# B&R Automation Studio project YuMiLAB_project (part 2)

#### Main.c
```c
// ************************************************************************************************************************************ //
// Title: Data processing -> Barcode Scanner
// Autor: Roman Parak
// Date : 8.5.2020
// Email: Roman.Parak@outlook.com
// ************************************************************************************************************************************ //

// ************************************************************************************************************************************ //
// -------------------------------------------------------------  LIBRARIES ----------------------------------------------------------- //
// ************************************************************************************************************************************ //
#include <bur/plctypes.h>

#ifdef _DEFAULT_INCLUDES
	#include <AsDefault.h>
#endif

#include <astime.h>

// ************************************************************************************************************************************ //
// -------------------------------------------------------------  DECLARATIONS -------------------------------------------------------- //
// ************************************************************************************************************************************ //
// BOOL
_LOCAL BOOL enable;
// UINT
_LOCAL UINT status;
_LOCAL UINT barcode_state;
// DATE_AND_TIME
_LOCAL DATE_AND_TIME DT1;
// DTGetTime_typ
_LOCAL DTGetTime_typ DTGetTime_1;
// INT
_LOCAL INT scan_counter;

// Declaration functions
void reset_data_mv();
void reset_data_init();

// ************************************************************************************************************************************ //
// -----------------------------------------------------------  INITIALIZATION -------------------------------------------------------- //
// ************************************************************************************************************************************ //
void _INIT ProgramInit(void)
{
	// Read/Write Data from Rpi
	(UDINT)strcpy(g_YuMiLab.scanner_m.rw_data_barcode.barcode_id, "");
	(UDINT)strcpy(g_YuMiLab.scanner_m.rw_data_barcode.tray_id, "");

	// Barcode parameters
	g_YuMiLab.scanner_m.rw_data_barcode.command    = 0;
	g_YuMiLab.scanner_m.rw_data_barcode.error_code = 0;
	g_YuMiLab.scanner_m.rw_data_barcode.barcode_scanner_module_ok = 0;
	g_YuMiLab.scanner_m.rw_data_barcode.tray_position_column = 3;
	g_YuMiLab.scanner_m.rw_data_barcode.tray_position_row    = 4;

	// Actual Data
	(UDINT)strcpy(g_YuMiLab.scanner_m.actual_barcode_id, "");
	(UDINT)strcpy(g_YuMiLab.scanner_m.actual_tray_id, "");

	// Data MappView {history} -> Initialization
	reset_data_mv();

	// FeID set/reset
	g_YuMiLab.scanner_m.feid_cmd_str.set = 0;
	g_YuMiLab.scanner_m.feid_cmd_str.reset = 0;
	g_YuMiLab.scanner_m.feid_cmd_str.enable_mv = 1;

	// Feid command
	(UDINT)strcpy(g_YuMiLab.scanner_m.feid_cmd_str.tray_id,"");

	// Main State
	barcode_state = 0;

	// Scan counter
	scan_counter = 0;
}

// ************************************************************************************************************************************ //
// -----------------------------------------------------------  MAIN (Cyclic) --------------------------------------------------------- //
// ************************************************************************************************************************************ //
void _CYCLIC ProgramCyclic(void)
{

	switch(barcode_state){
		case 0:
			{
				/*************************************** INITIALIZATION STATE ******************************************/

				// err-states:
				/*
				ok = 0
				eID_not_in_database = 1
				tray_warning_FeID_used = 2  # no new DB entry added for sample_tray, using existing
				tray_not_created = 3  # cannot add new sample_tray
				tray_position_not_assigned = 4
				service_connection_lost = 5  # cannot access DB
				*/
				// cmd {0} -> nothing ok, cmd {1} - write FeID , cmd {2} -> scan, cmd {3} ->  write row, column

				//(UDINT)strcpy(g_YuMiLab.scanner_m.rw_data_barcode.barcode_id, "");

				// reset scan err.
				g_YuMiLab.scanner_m.scan_err = 0;

				// Copy
				g_YuMiLab.scanner_m.cmd.write_FeID = g_YuMiLab.scanner_m.feid_cmd_str.set;

				// Condition -> Scanner module is ok!
				if(g_YuMiLab.scanner_m.rw_data_barcode.barcode_scanner_module_ok == 1){
					// reset error code
					g_YuMiLab.scanner_m.rw_data_barcode.error_code = 0;

					if(g_YuMiLab.scanner_m.cmd.write_FeID == 1){
						//cmd {1} - write FeID
						barcode_state = 1;
					}else if(g_YuMiLab.scanner_m.cmd.scan == 1){
						//cmd {2} -> scan
						(UDINT)strcpy(g_YuMiLab.scanner_m.rw_data_barcode.barcode_id, "None");
						// change state
						barcode_state = 3;
					}
				}
			}
			break;

		case 1:
			{
				/*************************************** WRITE FEID (1) STATE ******************************************/
				// reset write (Feid) command
				g_YuMiLab.scanner_m.cmd.write_FeID = 0;

				// mappview -> enable
				g_YuMiLab.scanner_m.feid_cmd_str.enable_mv = 0;

				// copy string
				(UDINT)strcpy(g_YuMiLab.scanner_m.actual_tray_id ,g_YuMiLab.scanner_m.feid_cmd_str.tray_id);
				(UDINT)strcpy(g_YuMiLab.scanner_m.rw_data_barcode.tray_id,g_YuMiLab.scanner_m.feid_cmd_str.tray_id);

				// command set -> 1
				g_YuMiLab.scanner_m.rw_data_barcode.command = 1;

				// change state -> check result
				barcode_state = 2;

			}
			break;
		case 2:
			{
				/*************************************** WRITE FEID (1a) STATE ******************************************/
				// Err. Condition -> module, err. code -> see bellow (info)
				if(g_YuMiLab.scanner_m.rw_data_barcode.barcode_scanner_module_ok == 0 || g_YuMiLab.scanner_m.rw_data_barcode.error_code > 0){
					// err. state var.
					err_state_barcode = 1;
					// command -> null
					g_YuMiLab.scanner_m.rw_data_barcode.command = 0;
					// change state -> initialization
					barcode_state = 0;
				}

				// Condition -> cmd null
				if(g_YuMiLab.scanner_m.rw_data_barcode.command == 0){
					// change state -> initialization
					barcode_state = 0;
				}
			}
			break;
		case 3:
			{
				/*************************************** START SCAN (1) STATE ******************************************/

				// scan var. -> null
				g_YuMiLab.scanner_m.cmd.scan = 0;

				// command -> 2
				g_YuMiLab.scanner_m.rw_data_barcode.command = 2;

				// changa state
				barcode_state = 4;

				// Err. Condition -> module
				if(g_YuMiLab.scanner_m.rw_data_barcode.barcode_scanner_module_ok == 0){
					// err. state var.
					err_state_barcode = 1;
					// command -> null
					g_YuMiLab.scanner_m.rw_data_barcode.command = 0;
					// change state -> initialization
					barcode_state = 0;
				}
			}
			break;

		case 4:
			{
				/*************************************** START SCAN (1a) STATE ******************************************/

				if(g_YuMiLab.scanner_m.rw_data_barcode.command == 0){
					//cmd {3} -> write row, column
					barcode_state = 5;
				}else if(g_YuMiLab.scanner_m.rw_data_barcode.error_code > 0 || (barcode_scan_state_next == 1 && g_YuMiLab.scanner_m.rw_data_barcode.command > 0)){
					// Err. Condition -> module, err. code -> see bellow (info)
					// err. state var.
					err_state_barcode = 1;
					// command -> null
					g_YuMiLab.scanner_m.rw_data_barcode.command = 0;

					// continue
					barcode_state = 5;
				}
			}
			break;
		case 5:
			{
				/*************************************** START SCAN (2) STATE ******************************************/

				// read barcode id
				(UDINT)strcpy(g_YuMiLab.scanner_m.actual_barcode_id , g_YuMiLab.scanner_m.rw_data_barcode.barcode_id);
				// write to table
				(UDINT)strcpy(g_YuMiLab.scanner_m.data_mv.barcode_id[scan_counter],g_YuMiLab.scanner_m.rw_data_barcode.barcode_id);
				// write column, row -> index of the current barcode ID
				g_YuMiLab.scanner_m.rw_data_barcode.tray_position_column = g_YuMiLab.scanner_m.data_mv.index_column[scan_counter];
				g_YuMiLab.scanner_m.rw_data_barcode.tray_position_row    = g_YuMiLab.scanner_m.data_mv.index_row[scan_counter];

				// Get actual time
				DTGetTime_1.enable = 1;
				// Call function
				DTGetTime(&DTGetTime_1);
				// Write time to the table
				ascDT(DTGetTime_1.DT1,(UDINT)&g_YuMiLab.scanner_m.data_mv.time[scan_counter], 128);

				// turn off function block
				DTGetTime_1.enable = 0;

				// Err. Condition -> err. code
				if(g_YuMiLab.scanner_m.rw_data_barcode.error_code > 0){
					// err. state var.
					err_state_barcode = 1;
					// error info -> with current index
					g_YuMiLab.scanner_m.data_mv.err_info[scan_counter] = 1;
				}

				// command -> 3
				g_YuMiLab.scanner_m.rw_data_barcode.command = 3;

				// change state
				barcode_state = 6;

			}
			break;

		case 6:
			{
				/*************************************** START SCAN (3) STATE ******************************************/

				// Err. Condition -> module, err. code -> see bellow (info)
				if(g_YuMiLab.scanner_m.rw_data_barcode.barcode_scanner_module_ok == 0 || g_YuMiLab.scanner_m.rw_data_barcode.error_code > 0){
					// err. state var.
					err_state_barcode = 1;

					// check counter max var.
					if(scan_counter < 11){
						// increase var. + 1
						scan_counter = scan_counter + 1;
					}else {
						// reset counter
						scan_counter = 0;
					}

					// command -> null
					g_YuMiLab.scanner_m.rw_data_barcode.command = 0;

					// change state -> initialization
					barcode_state = 0;
				}else{

					// Condition -> Command null (info from barcode app.)?
					if(g_YuMiLab.scanner_m.rw_data_barcode.command == 0){
						// check counter max var.
						if(scan_counter < 11){
							// increase var. + 1
							scan_counter = scan_counter + 1;
						}else {
							// reset counter
							scan_counter = 0;
						}

						// change state -> initialization
						barcode_state = 0;
					}else if(barcode_scan_state_next == 1 && g_YuMiLab.scanner_m.rw_data_barcode.command > 0){
						// Condition -> Command > 0 (no information from barcode app.) and aux. var from another task (Robot_m.c)
						// err. state var.
						err_state_barcode = 1;
						// command -> null
						g_YuMiLab.scanner_m.rw_data_barcode.command = 0;

						// check counter max var.
						if(scan_counter < 11){
							// increase var. + 1
							scan_counter = scan_counter + 1;
						}else {
							// reset counter
							scan_counter = 0;
						}

						// change state -> initialization
						barcode_state = 0;
					}
				}

				// Copy counter: Local var. -> Global var.
				g_YuMiLab.robot_m.counter = scan_counter;
			}
			break;
	}

	// function for reset current Feid
	if(g_YuMiLab.scanner_m.feid_cmd_str.reset == 1){
		// Feid -> null
		(UDINT)strcpy(g_YuMiLab.scanner_m.feid_cmd_str.tray_id,"");
		// enable textbox
		g_YuMiLab.scanner_m.feid_cmd_str.enable_mv = 1;
	}

	// reset mappview data
	if(g_YuMiLab.scanner_m.reset_data_mv == 1){
		// call function
		reset_data_init();
	}
}

// ************************************************************************************************************************************ //
// ------------------------------------------------------------  FUNCTIONS ------------------------------------------------------------ //
// ************************************************************************************************************************************ //

// **************** RESET DATA MAPPVIEW ********************** //
void reset_data_mv(){
	(UDINT)strcpy(g_YuMiLab.scanner_m.data_mv.barcode_id[0], "");
	(UDINT)strcpy(g_YuMiLab.scanner_m.data_mv.barcode_id[1], "");
	(UDINT)strcpy(g_YuMiLab.scanner_m.data_mv.barcode_id[2], "");
	(UDINT)strcpy(g_YuMiLab.scanner_m.data_mv.barcode_id[3], "");
	(UDINT)strcpy(g_YuMiLab.scanner_m.data_mv.barcode_id[4], "");
	(UDINT)strcpy(g_YuMiLab.scanner_m.data_mv.barcode_id[5], "");
	(UDINT)strcpy(g_YuMiLab.scanner_m.data_mv.barcode_id[6], "");
	(UDINT)strcpy(g_YuMiLab.scanner_m.data_mv.barcode_id[7], "");
	(UDINT)strcpy(g_YuMiLab.scanner_m.data_mv.barcode_id[8], "");
	(UDINT)strcpy(g_YuMiLab.scanner_m.data_mv.barcode_id[9], "");
	(UDINT)strcpy(g_YuMiLab.scanner_m.data_mv.barcode_id[10], "");
	(UDINT)strcpy(g_YuMiLab.scanner_m.data_mv.barcode_id[11], "");

	(UDINT)strcpy(g_YuMiLab.scanner_m.data_mv.time[0], "");
	(UDINT)strcpy(g_YuMiLab.scanner_m.data_mv.time[1], "");
	(UDINT)strcpy(g_YuMiLab.scanner_m.data_mv.time[2], "");
	(UDINT)strcpy(g_YuMiLab.scanner_m.data_mv.time[3], "");
	(UDINT)strcpy(g_YuMiLab.scanner_m.data_mv.time[4], "");
	(UDINT)strcpy(g_YuMiLab.scanner_m.data_mv.time[5], "");
	(UDINT)strcpy(g_YuMiLab.scanner_m.data_mv.time[6], "");
	(UDINT)strcpy(g_YuMiLab.scanner_m.data_mv.time[7], "");
	(UDINT)strcpy(g_YuMiLab.scanner_m.data_mv.time[8], "");
	(UDINT)strcpy(g_YuMiLab.scanner_m.data_mv.time[9], "");
	(UDINT)strcpy(g_YuMiLab.scanner_m.data_mv.time[10], "");
	(UDINT)strcpy(g_YuMiLab.scanner_m.data_mv.time[11], "");

	g_YuMiLab.scanner_m.data_mv.err_info[0] = 0;
	g_YuMiLab.scanner_m.data_mv.err_info[1] = 0;
	g_YuMiLab.scanner_m.data_mv.err_info[2] = 0;
	g_YuMiLab.scanner_m.data_mv.err_info[3] = 0;
	g_YuMiLab.scanner_m.data_mv.err_info[4] = 0;
	g_YuMiLab.scanner_m.data_mv.err_info[5] = 0;
	g_YuMiLab.scanner_m.data_mv.err_info[6] = 0;
	g_YuMiLab.scanner_m.data_mv.err_info[7] = 0;
	g_YuMiLab.scanner_m.data_mv.err_info[8] = 0;
	g_YuMiLab.scanner_m.data_mv.err_info[9] = 0;
	g_YuMiLab.scanner_m.data_mv.err_info[10] = 0;
	g_YuMiLab.scanner_m.data_mv.err_info[11] = 0;

	g_YuMiLab.scanner_m.data_mv.index[0] = 1;
	g_YuMiLab.scanner_m.data_mv.index[1] = 2;
	g_YuMiLab.scanner_m.data_mv.index[2] = 3;
	g_YuMiLab.scanner_m.data_mv.index[3] = 4;
	g_YuMiLab.scanner_m.data_mv.index[4] = 5;
	g_YuMiLab.scanner_m.data_mv.index[5] = 6;
	g_YuMiLab.scanner_m.data_mv.index[6] = 7;
	g_YuMiLab.scanner_m.data_mv.index[7] = 8;
	g_YuMiLab.scanner_m.data_mv.index[8] = 9;
	g_YuMiLab.scanner_m.data_mv.index[9] = 10;
	g_YuMiLab.scanner_m.data_mv.index[10] = 11;
	g_YuMiLab.scanner_m.data_mv.index[11] = 12;

	g_YuMiLab.scanner_m.data_mv.index_column[0] = 1;
	g_YuMiLab.scanner_m.data_mv.index_column[1] = 2;
	g_YuMiLab.scanner_m.data_mv.index_column[2] = 3;
	g_YuMiLab.scanner_m.data_mv.index_column[3] = 1;
	g_YuMiLab.scanner_m.data_mv.index_column[4] = 2;
	g_YuMiLab.scanner_m.data_mv.index_column[5] = 3;
	g_YuMiLab.scanner_m.data_mv.index_column[6] = 1;
	g_YuMiLab.scanner_m.data_mv.index_column[7] = 2;
	g_YuMiLab.scanner_m.data_mv.index_column[8] = 3;
	g_YuMiLab.scanner_m.data_mv.index_column[9] = 1;
	g_YuMiLab.scanner_m.data_mv.index_column[10] = 2;
	g_YuMiLab.scanner_m.data_mv.index_column[11] = 3;

	g_YuMiLab.scanner_m.data_mv.index_row[0]    = 1;
	g_YuMiLab.scanner_m.data_mv.index_row[1]    = 1;
	g_YuMiLab.scanner_m.data_mv.index_row[2]    = 1;
	g_YuMiLab.scanner_m.data_mv.index_row[3]    = 2;
	g_YuMiLab.scanner_m.data_mv.index_row[4]    = 2;
	g_YuMiLab.scanner_m.data_mv.index_row[5]    = 2;
	g_YuMiLab.scanner_m.data_mv.index_row[6]    = 3;
	g_YuMiLab.scanner_m.data_mv.index_row[7]    = 3;
	g_YuMiLab.scanner_m.data_mv.index_row[8]    = 3;
	g_YuMiLab.scanner_m.data_mv.index_row[9]    = 4;
	g_YuMiLab.scanner_m.data_mv.index_row[10]   = 4;
	g_YuMiLab.scanner_m.data_mv.index_row[11]   = 4;
} // end function

// **************** RESET INITIALIZATION DATA ********************** //
void reset_data_init(){
	// Read/Write Data from Rpi
	(UDINT)strcpy(g_YuMiLab.scanner_m.rw_data_barcode.barcode_id, "");
	(UDINT)strcpy(g_YuMiLab.scanner_m.rw_data_barcode.tray_id, "");

	// Barcode parameters
	g_YuMiLab.scanner_m.rw_data_barcode.command    = 0;
	g_YuMiLab.scanner_m.rw_data_barcode.error_code = 0;
	g_YuMiLab.scanner_m.rw_data_barcode.barcode_scanner_module_ok = 0;
	g_YuMiLab.scanner_m.rw_data_barcode.tray_position_column = 3;
	g_YuMiLab.scanner_m.rw_data_barcode.tray_position_row    = 4;

	// Actual Data
	(UDINT)strcpy(g_YuMiLab.scanner_m.actual_barcode_id, "");
	(UDINT)strcpy(g_YuMiLab.scanner_m.actual_tray_id, "");

	// Data MappView {history} -> Initialization
	reset_data_mv();

	// FeID set/reset
	g_YuMiLab.scanner_m.feid_cmd_str.set = 0;
	g_YuMiLab.scanner_m.feid_cmd_str.reset = 0;
	g_YuMiLab.scanner_m.feid_cmd_str.enable_mv = 1;

	// Feid command
	(UDINT)strcpy(g_YuMiLab.scanner_m.feid_cmd_str.tray_id,"");

	// Main state
	barcode_state = 0;

	// Scan Counter
	scan_counter = 0;
} // end function
```

### Program Logical/Technology/Robot_m (ANSIC)

#### Main.c
```c
// ************************************************************************************************************************************ //
// Title: ABB Robot Control -> Input/Output
// Autor: Roman Parak
// Date : 8.5.2020
// Email: Roman.Parak@outlook.com
// ************************************************************************************************************************************ //

// ************************************************************************************************************************************ //
// -------------------------------------------------------------  LIBRARIES ----------------------------------------------------------- //
// ************************************************************************************************************************************ //
#include <bur/plctypes.h>

#ifdef _DEFAULT_INCLUDES
	#include <AsDefault.h>
#endif

// ************************************************************************************************************************************ //
// -------------------------------------------------------------  DECLARATIONS -------------------------------------------------------- //
// ************************************************************************************************************************************ //
// UINT
_LOCAL UINT robot_state;
// INT
_LOCAL INT robot_counter, before_robot_counter;
// BOOL
_LOCAL BOOL power_on_off, motor_on_off;
_LOCAL BOOL wTO_smc;

// DEFINE
#define SERVO_OPEN 790
#define SERVO_CLOSE 570
#define SERVO_OPEN_B 1000
#define SERVO_CLOSE_B 0

// Declaration functions
void reset_data_init();

// ************************************************************************************************************************************ //
// -----------------------------------------------------------  INITIALIZATION -------------------------------------------------------- //
// ************************************************************************************************************************************ //
void _INIT ProgramInit(void)
{
	// err. state var.
	err_state_barcode = 0;

	// aux. variable -> turn on/turn off smc tube opener
	wTO_smc = 0;

	// Tube opener -> default param. (mode)
	g_YuMiLab.tube_opener.actual_state.Mode.Attached = 0;
	g_YuMiLab.tube_opener.actual_state.Mode.Close 	 = 0;
	g_YuMiLab.tube_opener.actual_state.Mode.Detached = 0;
	g_YuMiLab.tube_opener.actual_state.Mode.Open 	 = 0;

	// Servo Cover -> default param. (pos., move)
	g_YuMiLab.servo_cover.Position = SERVO_OPEN;
	g_YuMiLab.servo_cover.cmd.Move = 1;

	// Robot Counter
	robot_counter = 0;

	// Before robot counter
	before_robot_counter = 0;

	// Main State
	robot_state = 0;
}

// ************************************************************************************************************************************ //
// -----------------------------------------------------------  MAIN (Cyclic) --------------------------------------------------------- //
// ************************************************************************************************************************************ //
void _CYCLIC ProgramCyclic(void)
{
	/*******************************************************************************************************************/
	/*********************************************** SIGNALIZATION NOTE ************************************************/
	/*******************************************************************************************************************/
	/*************************************** Wait 0, In Progress 1, Successful 2 ***************************************/
	/*******************************************************************************************************************/

	switch(robot_state){
		case 0:
			{
				/*************************************** Start Stage ***************************************/

				// ----------------------------------------------------------------------------------- //
				// -------------------- Write actual signalization of each states -------------------- //
				// ----------------------------------------------------------------------------------- //
				(UDINT)strcpy(g_YuMiLab.robot_m.info_stage.Stage_1_TubeR.Status_str, "Wait");
				g_YuMiLab.robot_m.info_stage.Stage_1_TubeR.Status_int = 0;

				(UDINT)strcpy(g_YuMiLab.robot_m.info_stage.Stage_2_Barcode.Status_str, "Wait");
				g_YuMiLab.robot_m.info_stage.Stage_2_Barcode.Status_int = 0;

				(UDINT)strcpy(g_YuMiLab.robot_m.info_stage.Stage_3_TubeO.Status_str, "Wait");
				g_YuMiLab.robot_m.info_stage.Stage_3_TubeO.Status_int = 0;

				(UDINT)strcpy(g_YuMiLab.robot_m.info_stage.Stage_4_PipR.Status_str, "Wait");
				g_YuMiLab.robot_m.info_stage.Stage_4_PipR.Status_int = 0;

				(UDINT)strcpy(g_YuMiLab.robot_m.info_stage.Stage_5_TroghP.Status_str, "Wait");
				g_YuMiLab.robot_m.info_stage.Stage_5_TroghP.Status_int = 0;

				(UDINT)strcpy(g_YuMiLab.robot_m.info_stage.Stage_6_Bin.Status_str, "Wait");
				g_YuMiLab.robot_m.info_stage.Stage_6_Bin.Status_int = 0;

				(UDINT)strcpy(g_YuMiLab.robot_m.info_stage.Stage_3_TubeO.Info, "Closed");
				// ----------------------------------------------------------------------------------- //
				// ----------------------------------------------------------------------------------- //
				// ----------------------------------------------------------------------------------- //

				//g_YuMiLab.robot_m.info_stage.Stage_1_TubeR.Info[robot_counter]  = 0;
				//g_YuMiLab.robot_m.info_stage.Stage_4_PipR.Info[robot_counter]   = 0;
				//g_YuMiLab.robot_m.info_stage.Stage_5_TroghP.Info[robot_counter] = 0;

			}
			break;
		case 1:
			{
				/*************************************** Pick Tube Stage {Rack} ***************************************/

				// error state barcode -> reset
				err_state_barcode       = 0;
				// barcode scan next -> reset
				barcode_scan_state_next = 0;

				// default mode -> reset
				g_YuMiLab.tube_opener.actual_state.Mode.Open  = 0;
				g_YuMiLab.tube_opener.actual_state.Mode.Close = 0;

				// Condition -> counter
				if(before_robot_counter < 12){
					// copy
					before_robot_counter = robot_counter;
				}else{
					// call function -> reset
					reset_data_init();
				}

				// // robot actual state (signalization)
				g_YuMiLab.robot_m.actual_sate.In_Progress = robot_counter + 1;
				g_YuMiLab.robot_m.actual_sate.Successful  = robot_counter;
				g_YuMiLab.robot_m.actual_sate.Wait 		  = 12 - (robot_counter + 1);

				//servo_position = 790;

				// Condition -> Servo Cover (open/close)
				if(g_YuMiLab.servo_cover.actual_state.inPosition == 1 && g_YuMiLab.servo_cover.Actual_Position != SERVO_OPEN_B){
					// set -> open position var.
					g_YuMiLab.servo_cover.Position = SERVO_OPEN;
					// move
					g_YuMiLab.servo_cover.cmd.Move = 1;
				}

				// reset var. tube oepenr -> detached
				g_YuMiLab.tube_opener.actual_state.Mode.Detached = 0;

				// ----------------------------------------------------------------------------------- //
				// -------------------- Write actual signalization of each states -------------------- //
				// ----------------------------------------------------------------------------------- //
				(UDINT)strcpy(g_YuMiLab.robot_m.info_stage.Stage_1_TubeR.Status_str, "In Progress");
				g_YuMiLab.robot_m.info_stage.Stage_1_TubeR.Status_int = 1;

				(UDINT)strcpy(g_YuMiLab.robot_m.info_stage.Stage_2_Barcode.Status_str, "Wait");
				g_YuMiLab.robot_m.info_stage.Stage_2_Barcode.Status_int = 0;

				(UDINT)strcpy(g_YuMiLab.robot_m.info_stage.Stage_3_TubeO.Status_str, "Wait");
				g_YuMiLab.robot_m.info_stage.Stage_3_TubeO.Status_int = 0;

				(UDINT)strcpy(g_YuMiLab.robot_m.info_stage.Stage_4_PipR.Status_str, "Wait");
				g_YuMiLab.robot_m.info_stage.Stage_4_PipR.Status_int = 0;

				(UDINT)strcpy(g_YuMiLab.robot_m.info_stage.Stage_5_TroghP.Status_str, "Wait");
				g_YuMiLab.robot_m.info_stage.Stage_5_TroghP.Status_int = 0;

				(UDINT)strcpy(g_YuMiLab.robot_m.info_stage.Stage_6_Bin.Status_str, "Wait");
				g_YuMiLab.robot_m.info_stage.Stage_6_Bin.Status_int = 0;
				// ----------------------------------------------------------------------------------- //
				// ----------------------------------------------------------------------------------- //
				// ----------------------------------------------------------------------------------- //

				// current sample -> info
				g_YuMiLab.robot_m.info_stage.Stage_1_TubeR.Info[robot_counter] = 1;

			}
			break;
		case 2:
			{
				/*************************************** Barcode Scan Stage  ***************************************/

				// ----------------------------------------------------------------------------------- //
				// -------------------- Write actual signalization of each states -------------------- //
				// ----------------------------------------------------------------------------------- //
				(UDINT)strcpy(g_YuMiLab.robot_m.info_stage.Stage_1_TubeR.Status_str, "Successful");
				g_YuMiLab.robot_m.info_stage.Stage_1_TubeR.Status_int = 2;

				(UDINT)strcpy(g_YuMiLab.robot_m.info_stage.Stage_2_Barcode.Status_str, "In Progress");
				g_YuMiLab.robot_m.info_stage.Stage_2_Barcode.Status_int = 1;

				(UDINT)strcpy(g_YuMiLab.robot_m.info_stage.Stage_3_TubeO.Status_str, "Wait");
				g_YuMiLab.robot_m.info_stage.Stage_3_TubeO.Status_int = 0;

				(UDINT)strcpy(g_YuMiLab.robot_m.info_stage.Stage_4_PipR.Status_str, "Wait");
				g_YuMiLab.robot_m.info_stage.Stage_4_PipR.Status_int = 0;

				(UDINT)strcpy(g_YuMiLab.robot_m.info_stage.Stage_5_TroghP.Status_str, "Wait");
				g_YuMiLab.robot_m.info_stage.Stage_5_TroghP.Status_int = 0;

				(UDINT)strcpy(g_YuMiLab.robot_m.info_stage.Stage_6_Bin.Status_str, "Wait");
				g_YuMiLab.robot_m.info_stage.Stage_6_Bin.Status_int = 0;
				// ----------------------------------------------------------------------------------- //
				// ----------------------------------------------------------------------------------- //
				// ----------------------------------------------------------------------------------- //

				// current sample -> info
				g_YuMiLab.robot_m.info_stage.Stage_1_TubeR.Info[robot_counter] = 2;

			}
			break;
		case 3:
			{
				/*************************************** Place Tube Stage {Tube Opener} ***************************************/

				//servo_position = 570;

				// Condition -> Servo Cover (open/close)
				if(g_YuMiLab.servo_cover.actual_state.inPosition == 1 && g_YuMiLab.servo_cover.Actual_Position != SERVO_CLOSE_B){
					// set -> open position var.
					g_YuMiLab.servo_cover.Position = SERVO_CLOSE;
					// move
					g_YuMiLab.servo_cover.cmd.Move = 1;
				}

				// ----------------------------------------------------------------------------------- //
				// -------------------- Write actual signalization of each states -------------------- //
				// ----------------------------------------------------------------------------------- //
				(UDINT)strcpy(g_YuMiLab.robot_m.info_stage.Stage_1_TubeR.Status_str, "Successful");
				g_YuMiLab.robot_m.info_stage.Stage_1_TubeR.Status_int = 2;

				(UDINT)strcpy(g_YuMiLab.robot_m.info_stage.Stage_2_Barcode.Status_str, "Successful");
				g_YuMiLab.robot_m.info_stage.Stage_2_Barcode.Status_int = 2;

				(UDINT)strcpy(g_YuMiLab.robot_m.info_stage.Stage_3_TubeO.Status_str, "In Progress");
				g_YuMiLab.robot_m.info_stage.Stage_3_TubeO.Status_int = 1;

				(UDINT)strcpy(g_YuMiLab.robot_m.info_stage.Stage_4_PipR.Status_str, "Wait");
				g_YuMiLab.robot_m.info_stage.Stage_4_PipR.Status_int = 0;

				(UDINT)strcpy(g_YuMiLab.robot_m.info_stage.Stage_5_TroghP.Status_str, "Wait");
				g_YuMiLab.robot_m.info_stage.Stage_5_TroghP.Status_int = 0;

				(UDINT)strcpy(g_YuMiLab.robot_m.info_stage.Stage_6_Bin.Status_str, "Wait");
				g_YuMiLab.robot_m.info_stage.Stage_6_Bin.Status_int = 0;
				// ----------------------------------------------------------------------------------- //
				// ----------------------------------------------------------------------------------- //
				// ----------------------------------------------------------------------------------- //

			}
			break;
		case 4:
			{
				/*************************************** Pick Pipette Stage  ***************************************/

				// open tube
				g_YuMiLab.tube_opener.cmd.Mode.Open_T = 1;

				//servo_position = 0;

				// mode -> attached
				g_YuMiLab.tube_opener.actual_state.Mode.Attached = 0;

				// ----------------------------------------------------------------------------------- //
				// -------------------- Write actual signalization of each states -------------------- //
				// ----------------------------------------------------------------------------------- //
				(UDINT)strcpy(g_YuMiLab.robot_m.info_stage.Stage_3_TubeO.Info, "Open");

				(UDINT)strcpy(g_YuMiLab.robot_m.info_stage.Stage_1_TubeR.Status_str, "Successful");
				g_YuMiLab.robot_m.info_stage.Stage_1_TubeR.Status_int = 2;

				(UDINT)strcpy(g_YuMiLab.robot_m.info_stage.Stage_2_Barcode.Status_str, "Successful");
				g_YuMiLab.robot_m.info_stage.Stage_2_Barcode.Status_int = 2;

				(UDINT)strcpy(g_YuMiLab.robot_m.info_stage.Stage_3_TubeO.Status_str, "Successful");
				g_YuMiLab.robot_m.info_stage.Stage_3_TubeO.Status_int = 2;

				(UDINT)strcpy(g_YuMiLab.robot_m.info_stage.Stage_4_PipR.Status_str, "In Progress");
				g_YuMiLab.robot_m.info_stage.Stage_4_PipR.Status_int = 1;

				(UDINT)strcpy(g_YuMiLab.robot_m.info_stage.Stage_5_TroghP.Status_str, "Wait");
				g_YuMiLab.robot_m.info_stage.Stage_5_TroghP.Status_int = 0;

				(UDINT)strcpy(g_YuMiLab.robot_m.info_stage.Stage_6_Bin.Status_str, "Wait");
				g_YuMiLab.robot_m.info_stage.Stage_6_Bin.Status_int = 0;
				// ----------------------------------------------------------------------------------- //
				// ----------------------------------------------------------------------------------- //
				// ----------------------------------------------------------------------------------- //

				// current sample -> info
				g_YuMiLab.robot_m.info_stage.Stage_4_PipR.Info[robot_counter] = 1;

				// barcode scan -> set next
				barcode_scan_state_next = 1;
			}
			break;
		case 5:
			{
				/*************************************** Place Pipette Stage {Tube Opener} ***************************************/

				// ----------------------------------------------------------------------------------- //
				// -------------------- Write actual signalization of each states -------------------- //
				// ----------------------------------------------------------------------------------- //
				(UDINT)strcpy(g_YuMiLab.robot_m.info_stage.Stage_1_TubeR.Status_str, "Successful");
				g_YuMiLab.robot_m.info_stage.Stage_1_TubeR.Status_int = 2;

				(UDINT)strcpy(g_YuMiLab.robot_m.info_stage.Stage_2_Barcode.Status_str, "Successful");
				g_YuMiLab.robot_m.info_stage.Stage_2_Barcode.Status_int = 2;

				(UDINT)strcpy(g_YuMiLab.robot_m.info_stage.Stage_3_TubeO.Status_str, "In Progress");
				g_YuMiLab.robot_m.info_stage.Stage_3_TubeO.Status_int = 1;

				(UDINT)strcpy(g_YuMiLab.robot_m.info_stage.Stage_4_PipR.Status_str, "Successful");
				g_YuMiLab.robot_m.info_stage.Stage_4_PipR.Status_int = 2;

				(UDINT)strcpy(g_YuMiLab.robot_m.info_stage.Stage_5_TroghP.Status_str, "Wait");
				g_YuMiLab.robot_m.info_stage.Stage_5_TroghP.Status_int = 0;

				(UDINT)strcpy(g_YuMiLab.robot_m.info_stage.Stage_6_Bin.Status_str, "Wait");
				g_YuMiLab.robot_m.info_stage.Stage_6_Bin.Status_int = 0;
				// ----------------------------------------------------------------------------------- //
				// ----------------------------------------------------------------------------------- //
				// ----------------------------------------------------------------------------------- //

				// current sample -> info
				g_YuMiLab.robot_m.info_stage.Stage_4_PipR.Info[robot_counter] = 2;

			}
			break;
		case 6:
			{
				/*************************************** Place Pipette Stage {Sample Tray} ***************************************/
				//servo_position = 790;

				// Condition -> Servo Cover (open/close)
				if(g_YuMiLab.servo_cover.actual_state.inPosition == 1 && g_YuMiLab.servo_cover.Actual_Position != SERVO_OPEN_B){
					// set -> open position var.
					g_YuMiLab.servo_cover.Position = SERVO_OPEN;
					// move
					g_YuMiLab.servo_cover.cmd.Move = 1;
				}

				// tube opener -> close
				g_YuMiLab.tube_opener.cmd.Mode.Closed_T = 1;
				// ----------------------------------------------------------------------------------- //
				// -------------------- Write actual signalization of each states -------------------- //
				// ----------------------------------------------------------------------------------- //
				(UDINT)strcpy(g_YuMiLab.robot_m.info_stage.Stage_1_TubeR.Status_str, "Successful");
				g_YuMiLab.robot_m.info_stage.Stage_1_TubeR.Status_int = 2;

				(UDINT)strcpy(g_YuMiLab.robot_m.info_stage.Stage_2_Barcode.Status_str, "Successful");
				g_YuMiLab.robot_m.info_stage.Stage_2_Barcode.Status_int = 2;

				(UDINT)strcpy(g_YuMiLab.robot_m.info_stage.Stage_3_TubeO.Status_str, "Successful");
				g_YuMiLab.robot_m.info_stage.Stage_3_TubeO.Status_int = 2;

				(UDINT)strcpy(g_YuMiLab.robot_m.info_stage.Stage_4_PipR.Status_str, "Successful");
				g_YuMiLab.robot_m.info_stage.Stage_4_PipR.Status_int = 2;

				(UDINT)strcpy(g_YuMiLab.robot_m.info_stage.Stage_5_TroghP.Status_str, "In Progress");
				g_YuMiLab.robot_m.info_stage.Stage_5_TroghP.Status_int = 1;

				(UDINT)strcpy(g_YuMiLab.robot_m.info_stage.Stage_6_Bin.Status_str, "Wait");
				g_YuMiLab.robot_m.info_stage.Stage_6_Bin.Status_int = 0;
				// ----------------------------------------------------------------------------------- //
				// ----------------------------------------------------------------------------------- //
				// ----------------------------------------------------------------------------------- //

				// current sample -> info
				g_YuMiLab.robot_m.info_stage.Stage_5_TroghP.Info[robot_counter] = 1;

			}
			break;
		case 7:
			{
				/*************************************** Place Pipette Stage {Bin} ***************************************/
				//servo_position = 570;

				// Condition -> Servo Cover (open/close)
				if(g_YuMiLab.servo_cover.actual_state.inPosition == 1 && g_YuMiLab.servo_cover.Actual_Position != SERVO_CLOSE_B){
					// set -> open position var.
					g_YuMiLab.servo_cover.Position = SERVO_CLOSE;
					// move
					g_YuMiLab.servo_cover.cmd.Move = 1;
				}

				// ----------------------------------------------------------------------------------- //
				// -------------------- Write actual signalization of each states -------------------- //
				// ----------------------------------------------------------------------------------- //
				(UDINT)strcpy(g_YuMiLab.robot_m.info_stage.Stage_3_TubeO.Info, "Closed");

				(UDINT)strcpy(g_YuMiLab.robot_m.info_stage.Stage_1_TubeR.Status_str, "Wait");
				g_YuMiLab.robot_m.info_stage.Stage_1_TubeR.Status_int = 0;

				(UDINT)strcpy(g_YuMiLab.robot_m.info_stage.Stage_2_Barcode.Status_str, "Successful");
				g_YuMiLab.robot_m.info_stage.Stage_2_Barcode.Status_int = 2;

				(UDINT)strcpy(g_YuMiLab.robot_m.info_stage.Stage_3_TubeO.Status_str, "Wait");
				g_YuMiLab.robot_m.info_stage.Stage_3_TubeO.Status_int = 0;

				(UDINT)strcpy(g_YuMiLab.robot_m.info_stage.Stage_4_PipR.Status_str, "Successful");
				g_YuMiLab.robot_m.info_stage.Stage_4_PipR.Status_int = 2;

				(UDINT)strcpy(g_YuMiLab.robot_m.info_stage.Stage_5_TroghP.Status_str, "Successful");
				g_YuMiLab.robot_m.info_stage.Stage_5_TroghP.Status_int = 2;

				(UDINT)strcpy(g_YuMiLab.robot_m.info_stage.Stage_6_Bin.Status_str, "In Progres");
				g_YuMiLab.robot_m.info_stage.Stage_6_Bin.Status_int = 1;
				// ----------------------------------------------------------------------------------- //
				// ----------------------------------------------------------------------------------- //
				// ----------------------------------------------------------------------------------- //

				// increase counter
				g_YuMiLab.robot_m.info_stage.Stage_6_Bin.Info = robot_counter + 1;

				// current sample -> info
				g_YuMiLab.robot_m.info_stage.Stage_5_TroghP.Info[robot_counter] = 2;

			}
			break;
		case 8:
			{
				/*************************************** Pick Tube Stage {Tube Opener} ***************************************/

				//servo_position = 0;

				// ----------------------------------------------------------------------------------- //
				// -------------------- Write actual signalization of each states -------------------- //
				// ----------------------------------------------------------------------------------- //
				(UDINT)strcpy(g_YuMiLab.robot_m.info_stage.Stage_1_TubeR.Status_str, "Wait");
				g_YuMiLab.robot_m.info_stage.Stage_1_TubeR.Status_int = 0;

				(UDINT)strcpy(g_YuMiLab.robot_m.info_stage.Stage_2_Barcode.Status_str, "Successful");
				g_YuMiLab.robot_m.info_stage.Stage_2_Barcode.Status_int = 2;

				(UDINT)strcpy(g_YuMiLab.robot_m.info_stage.Stage_3_TubeO.Status_str, "In Progres");
				g_YuMiLab.robot_m.info_stage.Stage_3_TubeO.Status_int = 1;

				(UDINT)strcpy(g_YuMiLab.robot_m.info_stage.Stage_4_PipR.Status_str, "Successful");
				g_YuMiLab.robot_m.info_stage.Stage_4_PipR.Status_int = 2;

				(UDINT)strcpy(g_YuMiLab.robot_m.info_stage.Stage_5_TroghP.Status_str, "Successful");
				g_YuMiLab.robot_m.info_stage.Stage_5_TroghP.Status_int = 2;

				(UDINT)strcpy(g_YuMiLab.robot_m.info_stage.Stage_6_Bin.Status_str, "Successful");
				g_YuMiLab.robot_m.info_stage.Stage_6_Bin.Status_int = 2;
				// ----------------------------------------------------------------------------------- //
				// ----------------------------------------------------------------------------------- //
				// ----------------------------------------------------------------------------------- //
			}
			break;
		case 9:
			{
				/*************************************** Place Tube Stage {Rack} ***************************************/

				// ----------------------------------------------------------------------------------- //
				// -------------------- Write actual signalization of each states -------------------- //
				// ----------------------------------------------------------------------------------- //
				(UDINT)strcpy(g_YuMiLab.robot_m.info_stage.Stage_1_TubeR.Status_str, "In Progres");
				g_YuMiLab.robot_m.info_stage.Stage_1_TubeR.Status_int = 1;

				(UDINT)strcpy(g_YuMiLab.robot_m.info_stage.Stage_2_Barcode.Status_str, "Successful");
				g_YuMiLab.robot_m.info_stage.Stage_2_Barcode.Status_int = 2;

				(UDINT)strcpy(g_YuMiLab.robot_m.info_stage.Stage_3_TubeO.Status_str, "Successful");
				g_YuMiLab.robot_m.info_stage.Stage_3_TubeO.Status_int = 2;

				(UDINT)strcpy(g_YuMiLab.robot_m.info_stage.Stage_4_PipR.Status_str, "Successful");
				g_YuMiLab.robot_m.info_stage.Stage_4_PipR.Status_int = 2;

				(UDINT)strcpy(g_YuMiLab.robot_m.info_stage.Stage_5_TroghP.Status_str, "Successful");
				g_YuMiLab.robot_m.info_stage.Stage_5_TroghP.Status_int = 2;

				(UDINT)strcpy(g_YuMiLab.robot_m.info_stage.Stage_6_Bin.Status_str, "Successful");
				g_YuMiLab.robot_m.info_stage.Stage_6_Bin.Status_int = 2;
				// ----------------------------------------------------------------------------------- //
				// ----------------------------------------------------------------------------------- //
				// ----------------------------------------------------------------------------------- //

				// -------------------- Counter ++ Stage -------------------- //

				// Condition -> set err. to current sample
				if(err_state_barcode == 1){
					// sample info
					g_YuMiLab.robot_m.info_stage.Stage_1_TubeR.Info[robot_counter]  = 3;
					g_YuMiLab.robot_m.info_stage.Stage_4_PipR.Info[robot_counter]   = 3;
					g_YuMiLab.robot_m.info_stage.Stage_5_TroghP.Info[robot_counter] = 3;

					// reset err. state
					err_state_barcode = 0;
				}

				// reset mode -> null
				g_YuMiLab.tube_opener.cmd.Mode.Open_T   = 0;
				g_YuMiLab.tube_opener.cmd.Mode.Closed_T = 0;

				//robot_counter = g_YuMiLab.robot_m.counter;

				if(before_robot_counter == robot_counter){
					// increase counter -> +1
					robot_counter = robot_counter + 1;
				}
			}
			break;
		case 10:
			{
				/*************************************** Pick Tube Stage {Rack} ***************************************/

				// ----------------------------------------------------------------------------------- //
				// -------------------- Write actual signalization of each states -------------------- //
				// ----------------------------------------------------------------------------------- //
				(UDINT)strcpy(g_YuMiLab.robot_m.info_stage.Stage_1_TubeR.Status_str, "Successful");
				g_YuMiLab.robot_m.info_stage.Stage_1_TubeR.Status_int = 2;

				(UDINT)strcpy(g_YuMiLab.robot_m.info_stage.Stage_2_Barcode.Status_str, "Successful");
				g_YuMiLab.robot_m.info_stage.Stage_2_Barcode.Status_int = 2;

				(UDINT)strcpy(g_YuMiLab.robot_m.info_stage.Stage_3_TubeO.Status_str, "Successful");
				g_YuMiLab.robot_m.info_stage.Stage_3_TubeO.Status_int = 2;

				(UDINT)strcpy(g_YuMiLab.robot_m.info_stage.Stage_4_PipR.Status_str, "Successful");
				g_YuMiLab.robot_m.info_stage.Stage_4_PipR.Status_int = 2;

				(UDINT)strcpy(g_YuMiLab.robot_m.info_stage.Stage_5_TroghP.Status_str, "Successful");
				g_YuMiLab.robot_m.info_stage.Stage_5_TroghP.Status_int = 2;

				(UDINT)strcpy(g_YuMiLab.robot_m.info_stage.Stage_6_Bin.Status_str, "Successful");
				g_YuMiLab.robot_m.info_stage.Stage_6_Bin.Status_int = 2;
				// ----------------------------------------------------------------------------------- //
				// ----------------------------------------------------------------------------------- //
				// ----------------------------------------------------------------------------------- //

			}
			break;
	}

	// turn on/turn off smc tube opener
	if(wTO_smc == 1){
		// attached
		g_YuMiLab.tube_opener.actual_state.Mode.Attached = 1;
		// close
		g_YuMiLab.tube_opener.actual_state.Mode.Close = 1;
		// detached
		g_YuMiLab.tube_opener.actual_state.Mode.Detached = 1;
		// open
		g_YuMiLab.tube_opener.actual_state.Mode.Open = 1;
	}

	// Condition -> Start: Power On is true
	if(power_on_off == 1){
		if(g_YuMiLab.robot_m.cmd.in_position_1 == 1){
			robot_state = 0;
		}else if(g_YuMiLab.robot_m.cmd.in_position_2 == 1){
			robot_state = 1;
		}else if(g_YuMiLab.robot_m.cmd.in_position_3 == 1){
			robot_state = 2;
		}else if(g_YuMiLab.robot_m.cmd.in_position_4 == 1){
			robot_state = 3;
		}else if(g_YuMiLab.robot_m.cmd.in_position_5 == 1){
			robot_state = 4;
		}else if(g_YuMiLab.robot_m.cmd.in_position_6 == 1){
			robot_state = 5;
		}else if(g_YuMiLab.robot_m.cmd.in_position_7 == 1){
			robot_state = 6;
		}else if(g_YuMiLab.robot_m.cmd.in_position_8 == 1){
			robot_state = 7;
		}else if(g_YuMiLab.robot_m.cmd.in_position_9 == 1){
			robot_state = 8;
		}else if(g_YuMiLab.robot_m.cmd.in_position_10 == 1){
			robot_state = 9;
		}
	}

	// Mappview -> Tube parameters Type 0, 1
	if(g_YuMiLab.robot_m.parameters_info.Tube.type == 0){
		g_YuMiLab.robot_m.parameters_info.Tube.param_a = 25;
		g_YuMiLab.robot_m.parameters_info.Tube.param_b = 20;
		g_YuMiLab.robot_m.parameters_info.Tube.param_c = 100;

		g_YuMiLab.robot_m.parameters_info.Tube.capacity = 7;
	}else if(g_YuMiLab.robot_m.parameters_info.Tube.type == 1){
		g_YuMiLab.robot_m.parameters_info.Tube.param_a = 10;
		g_YuMiLab.robot_m.parameters_info.Tube.param_b = 15;
		g_YuMiLab.robot_m.parameters_info.Tube.param_c = 75;

		g_YuMiLab.robot_m.parameters_info.Tube.capacity = 3;
	}

	// Mappview -> Pipette parameters Type 0, 1
	if(g_YuMiLab.robot_m.parameters_info.Pipette.type == 0){
		g_YuMiLab.robot_m.parameters_info.Pipette.param_a = 10;
		g_YuMiLab.robot_m.parameters_info.Pipette.param_b = 5;
		g_YuMiLab.robot_m.parameters_info.Pipette.param_c = 80;

		g_YuMiLab.robot_m.parameters_info.Pipette.capacity = 3;
	}else if(g_YuMiLab.robot_m.parameters_info.Pipette.type == 1){
		g_YuMiLab.robot_m.parameters_info.Pipette.param_a = 15;
		g_YuMiLab.robot_m.parameters_info.Pipette.param_b = 10;
		g_YuMiLab.robot_m.parameters_info.Pipette.param_c = 100;

		g_YuMiLab.robot_m.parameters_info.Pipette.capacity = 5;
	}

	// Power on/off robot ABB
	if(power_on_off == 1){
		g_YuMiLab.robot_m.cmd.power_off = 0;
		g_YuMiLab.robot_m.cmd.power_on  = 1;
	}else if(power_on_off == 0){
		robot_state = 0;
		g_YuMiLab.robot_m.cmd.power_on  = 0;
		g_YuMiLab.robot_m.cmd.power_off = 1;
	}

	// Motor on/off robot ABB
	if(g_YuMiLab.robot_m.actual_sate.is_motor_on == 1){
		motor_on_off = 1;
	}else if(g_YuMiLab.robot_m.actual_sate.is_motor_off == 1){
		motor_on_off = 0;
	}

	// reset mappview parameters
	if(g_YuMiLab.scanner_m.reset_data_mv == 1){
		reset_data_init();
	}
}

// ************************************************************************************************************************************ //
// ------------------------------------------------------------  FUNCTIONS ------------------------------------------------------------ //
// ************************************************************************************************************************************ //

// **************** RESET INITIALIZATION DATA ********************** //
void reset_data_init(){
	// robot actual state
	g_YuMiLab.robot_m.actual_sate.In_Progress = 0;
	g_YuMiLab.robot_m.actual_sate.Successful = 0;
	g_YuMiLab.robot_m.actual_sate.Wait = 0;

	// Robot Counter
	robot_counter = 0;

	// Before robot counter
	before_robot_counter = 0;

	// err. state var.
	err_state_barcode = 0;

	// -------------------- DEFAULT STR. SIGNALIZATION -------------------- //
	(UDINT)strcpy(g_YuMiLab.robot_m.info_stage.Stage_1_TubeR.Status_str, "Wait");
	g_YuMiLab.robot_m.info_stage.Stage_1_TubeR.Status_int = 0;

	(UDINT)strcpy(g_YuMiLab.robot_m.info_stage.Stage_2_Barcode.Status_str, "Wait");
	g_YuMiLab.robot_m.info_stage.Stage_2_Barcode.Status_int = 0;

	(UDINT)strcpy(g_YuMiLab.robot_m.info_stage.Stage_3_TubeO.Status_str, "Wait");
	g_YuMiLab.robot_m.info_stage.Stage_3_TubeO.Status_int = 0;

	(UDINT)strcpy(g_YuMiLab.robot_m.info_stage.Stage_4_PipR.Status_str, "Wait");
	g_YuMiLab.robot_m.info_stage.Stage_4_PipR.Status_int = 0;

	(UDINT)strcpy(g_YuMiLab.robot_m.info_stage.Stage_5_TroghP.Status_str, "Wait");
	g_YuMiLab.robot_m.info_stage.Stage_5_TroghP.Status_int = 0;

	(UDINT)strcpy(g_YuMiLab.robot_m.info_stage.Stage_6_Bin.Status_str, "Wait");
	g_YuMiLab.robot_m.info_stage.Stage_6_Bin.Status_int = 0;

	(UDINT)strcpy(g_YuMiLab.robot_m.info_stage.Stage_3_TubeO.Info, "Closed");

	g_YuMiLab.robot_m.info_stage.Stage_1_TubeR.Info[0] = 0;
	g_YuMiLab.robot_m.info_stage.Stage_1_TubeR.Info[1] = 0;
	g_YuMiLab.robot_m.info_stage.Stage_1_TubeR.Info[2] = 0;
	g_YuMiLab.robot_m.info_stage.Stage_1_TubeR.Info[3] = 0;
	g_YuMiLab.robot_m.info_stage.Stage_1_TubeR.Info[4] = 0;
	g_YuMiLab.robot_m.info_stage.Stage_1_TubeR.Info[5] = 0;
	g_YuMiLab.robot_m.info_stage.Stage_1_TubeR.Info[6] = 0;
	g_YuMiLab.robot_m.info_stage.Stage_1_TubeR.Info[7] = 0;
	g_YuMiLab.robot_m.info_stage.Stage_1_TubeR.Info[8] = 0;
	g_YuMiLab.robot_m.info_stage.Stage_1_TubeR.Info[9] = 0;
	g_YuMiLab.robot_m.info_stage.Stage_1_TubeR.Info[10] = 0;
	g_YuMiLab.robot_m.info_stage.Stage_1_TubeR.Info[11] = 0;

	g_YuMiLab.robot_m.info_stage.Stage_4_PipR.Info[0] = 0;
	g_YuMiLab.robot_m.info_stage.Stage_4_PipR.Info[1] = 0;
	g_YuMiLab.robot_m.info_stage.Stage_4_PipR.Info[2] = 0;
	g_YuMiLab.robot_m.info_stage.Stage_4_PipR.Info[3] = 0;
	g_YuMiLab.robot_m.info_stage.Stage_4_PipR.Info[4] = 0;
	g_YuMiLab.robot_m.info_stage.Stage_4_PipR.Info[5] = 0;
	g_YuMiLab.robot_m.info_stage.Stage_4_PipR.Info[6] = 0;
	g_YuMiLab.robot_m.info_stage.Stage_4_PipR.Info[7] = 0;
	g_YuMiLab.robot_m.info_stage.Stage_4_PipR.Info[8] = 0;
	g_YuMiLab.robot_m.info_stage.Stage_4_PipR.Info[9] = 0;
	g_YuMiLab.robot_m.info_stage.Stage_4_PipR.Info[10] = 0;
	g_YuMiLab.robot_m.info_stage.Stage_4_PipR.Info[11] = 0;

	g_YuMiLab.robot_m.info_stage.Stage_5_TroghP.Info[0] = 0;
	g_YuMiLab.robot_m.info_stage.Stage_5_TroghP.Info[1] = 0;
	g_YuMiLab.robot_m.info_stage.Stage_5_TroghP.Info[2] = 0;
	g_YuMiLab.robot_m.info_stage.Stage_5_TroghP.Info[3] = 0;
	g_YuMiLab.robot_m.info_stage.Stage_5_TroghP.Info[4] = 0;
	g_YuMiLab.robot_m.info_stage.Stage_5_TroghP.Info[5] = 0;
	g_YuMiLab.robot_m.info_stage.Stage_5_TroghP.Info[6] = 0;
	g_YuMiLab.robot_m.info_stage.Stage_5_TroghP.Info[7] = 0;
	g_YuMiLab.robot_m.info_stage.Stage_5_TroghP.Info[8] = 0;
	g_YuMiLab.robot_m.info_stage.Stage_5_TroghP.Info[9] = 0;
	g_YuMiLab.robot_m.info_stage.Stage_5_TroghP.Info[10] = 0;
	g_YuMiLab.robot_m.info_stage.Stage_5_TroghP.Info[11] = 0;
} // end function
```

### Program Logical/Technology/Tube_Opener (ANSIC)
